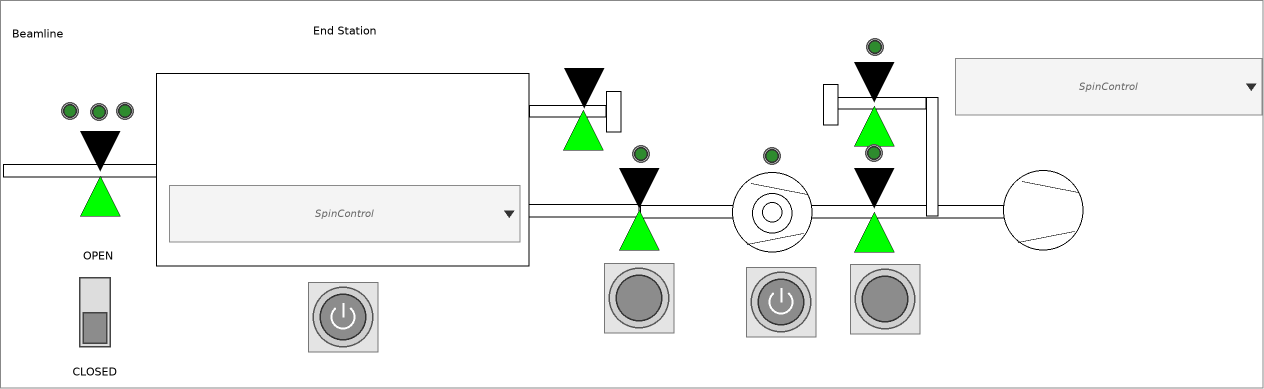
VISUALIZATION Vacuum  // 1264x389
    Rectangle (529,105 77x12)
    Rectangle (640,205 380x13), colour toggle: GVL_ver.VGC1_i_xDwstream_OK
    Rectangle (523,204 116x13), colour toggle: GVL_ver.VGC1_i_xUpstream_OK
    Rectangle (3,164 467x13)
    RoundedRectangle (156,73 373x193), colour toggle: GVL_ver.GCC1_xPRESS_OK
    SpinControl (169,185 351x57), variable: GVL_ver.GCC1_rPRESS
    SpinControl (955,58 307x57), variable: GVL_ver.GCC2_rPRESS
    PowerSwitch (308,282 70x70), variable: GVL_ver.GCC1_xHV_DIS, behaviour: TOGGLE, style: Switch-PowerSwitch-Gray
    PushSwitchLed (604,263 70x70), variable: GVL_ver.VGC1OPENREQ, behaviour: TOGGLE, style: Switch-PushSwitchLed-Gray
    Lamp1 (762,146 20x20), variable: GVL_ver.PTM1_i_xFaultNC, style: Lamp-Lamp1-Green
    PowerSwitch (746,267 70x70), variable: GVL_ver.PTM1STARTREQ, behaviour: TOGGLE, style: Switch-PowerSwitch-Gray
    Polygon (639,210) (639,210) (639,210) (659,250) (619,250), colour toggle: GVL_ver.VGC1_i_xClsLS
    Polygon (639,208) (639,208) (639,208) (659,168) (619,168), colour toggle: GVL_ver.VGC1_i_xOpnLS
    Ellipse (732,172 80x80), colour toggle: GVL_ver.PTM1_i_xAtSpd
    Ellipse (752,193 40x40), colour toggle: GVL_ver.PTM1_q_RunDO
    Ellipse (762,202 20x20), colour toggle: GVL_ver.PTM1_q_PumpingStation
    Polygon (874,208) (874,208) (874,208) (894,168) (854,168), colour toggle: GVL_ver.VCC2_i_xOpnLS
    Polygon (583,110) (583,110) (583,110) (603,150) (563,150), colour toggle: GVL_ver.VCC3_i_xClsLS
    PushSwitchLed (850,264 70x70), variable: GVL_ver.VCC2_r_OPENREQ, behaviour: TOGGLE, style: Switch-PushSwitchLed-Gray
    Line (822,135)
    Line (747,244) (803,233), colour toggle: GVL_ver.PTM1_q_xRemote
    Line (751,183) (807,194), colour toggle: GVL_ver.PTM1_i_xRemote
    Polygon (584,108) (584,108) (584,108) (604,68) (564,68), colour toggle: GVL_ver.VCC3_i_xOpnLS
    Rectangle (606,91 15x41)
    Polygon (100,171) (100,171) (100,171) (120,131) (80,131), colour toggle: GVL_ver.VGC0_i_xOpnLS
    Polygon (100,176) (100,176) (100,176) (120,216) (80,216), colour toggle: GVL_ver.VGC0_i_xClsLS
    Polygon (874,212) (874,212) (874,212) (894,252) (854,252), colour toggle: GVL_ver.VCC2_i_xClsLS
    Rectangle (824,97 102x12), colour toggle: GVL_ver.VGC1_i_xDwstream_OK
    Polygon (874,106) (874,106) (874,106) (894,146) (854,146), colour toggle: GVL_ver.VCC3_i_xClsLS
    Polygon (874,102) (874,102) (874,102) (894,62) (854,62), colour toggle: GVL_ver.VCC3_i_xOpnLS
    DipSwitch (60,277 70x70), variable: GVL_ver.VGC0OPENREQ, behaviour: TOGGLE, style: Switch-DipSwitch-Gray
    Label (63,241 70x30), "OPEN"
    Label (60,357 70x30), "CLOSED"
    Ellipse (1003,170 80x80), colour toggle: GVL_ver.PTM2_i_xAtSpd
    Line (1018,242) (1074,231), colour toggle: GVL_ver.PTM1_q_xRemote
    Line (1022,181) (1078,192), colour toggle: GVL_ver.PTM1_i_xRemote
    Rectangle (926,97 12x119), colour toggle: GVL_ver.VGC1_i_xDwstream_OK
    Rectangle (823,84 15x41)
    Label (3,19 70x30), "Beamline"
    Label (295,16 100x30), "End Station"
    Lamp1 (631,144 20x20), variable: GVL_ver.VGC1_q_xOPN_DO, style: Lamp-Lamp1-Green
    Lamp1 (89,102 20x20), variable: GVL_ver.VGC0_q_xOPN_DO, style: Lamp-Lamp1-Green
    Lamp1 (115,101 20x20), variable: GVL_ver.VGC0_i_xDwstream_OK, style: Lamp-Lamp1-Green
    Lamp1 (60,101 20x20), variable: GVL_ver.VGC0_i_xUpstream_OK, style: Lamp-Lamp1-Green
    Lamp1 (864,143 20x20), variable: GVL_ver.VCC2_q_xOPN_DO, style: Lamp-Lamp1-Green
    Lamp1 (865,37 20x20), variable: GVL_ver.VCC3_q_xOPN_DO, style: Lamp-Lamp1-Green
END_VISUALIZATION

(* stored: Version 1.1.0.1, ProductVersion 3.1.4022.3
   Visu Vacuum: Id {1073ae53-d0f5-4394-900f-79549f428b0f} *)
